Yaskawa INFORM job: CALIBRATION_RELATIVE.JBI

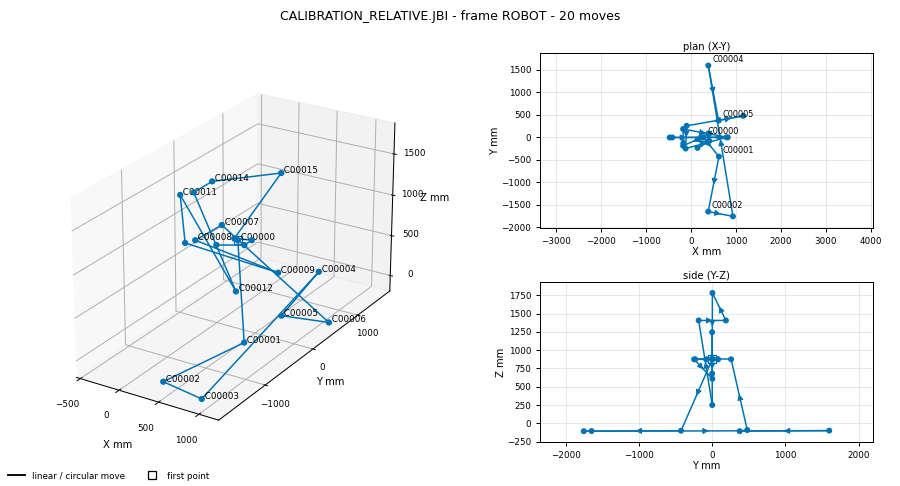
[picture p0: tool path of CALIBRATION_RELATIVE.JBI in frame ROBOT, 20 of 20 moves have a stored position in this frame; points joined in program order, loops and branches not executed]
/JOB
//NAME CALIBRATION_RELATIVE
//POS
///NPOS 20,0,0,0,0,0
///TOOL 0
///POSTYPE ROBOT
///RECTAN
///RCONF 1,0,0,0,0,0,0,0,0,0,0,0,0,0,0,0,0,0,0,0,0,0,0,0
C00000=274.980,-0.008,875.000,179.9989,44.9997,0.0020
C00001=622.573,-426.393,-101.139,-179.2940,-0.1745,-16.1282
C00002=383.550,-1649.719,-105.735,-178.5001,0.5026,-41.4095
C00003=933.399,-1756.204,-107.506,-178.6315,0.5025,-41.3677
C00004=385.503,1598.413,-99.610,-179.5797,-0.3013,-6.9319
C00005=613.623,374.870,-107.125,-179.5061,-0.2696,-6.9262
C00006=1163.774,478.153,-91.819,-179.4694,-0.2982,-6.9135
C00007=-96.141,257.633,874.999,180.0000,45.0002,110.4650
C00008=-118.644,-248.076,874.999,180.0000,45.0002,-115.5590
C00009=790.609,1.376,608.986,179.1795,83.3199,-0.7822
///RCONF 1,0,1,0,0,0,0,0,0,0,0,0,0,0,0,0,0,0,0,0,0,0,0,0
C00010=-414.668,-1.854,679.993,-179.8858,-2.8354,0.0446
C00011=-472.496,-2.009,1245.133,-179.8243,-31.5756,0.0258
///RCONF 1,0,0,0,0,0,0,0,0,0,0,0,0,0,0,0,0,0,0,0,0,0,0,0
C00012=249.873,-0.073,250.348,0.7052,79.6569,-179.2402
C00013=-173.865,-186.177,1406.145,147.2368,-45.5002,-134.7207
C00014=-174.385,186.529,1405.578,-146.8336,-45.3818,134.7676
///RCONF 0,0,0,0,0,0,0,0,0,0,0,0,0,0,0,0,0,0,0,0,0,0,0,0
C00015=818.445,1.458,1781.947,-6.0107,-88.9505,-173.7227
///RCONF 1,0,0,0,0,0,0,0,0,0,0,0,0,0,0,0,0,0,0,0,0,0,0,0
C00016=229.198,-0.125,884.124,179.9802,49.6969,-0.0171
///RCONF 1,0,0,0,1,0,0,0,0,0,0,0,0,0,0,0,0,0,0,0,0,0,0,0
C00017=404.652,79.634,874.999,179.9998,44.9999,-118.1512
C00018=406.759,-76.550,874.999,-179.9998,44.9999,118.4297
///RCONF 1,0,0,0,0,0,0,0,0,0,0,0,0,0,0,0,0,0,0,0,0,0,0,0
C00019=145.602,-233.286,874.998,180.0000,45.0007,-58.0294
//INST
///DATE 2026/08/24 08:52
///ATTR SC,RW,RJ
////FRAME ROBOT
///GROUP1 RB1
NOP
'1 HOME POSTION
MOVL C00000 V=423.3
'2 UF#2 S1 ORG
MOVL C00001 V=423.3
'3 UF#2 S1 RXX
MOVL C00002 V=423.3
'4 UF#2 S1 RXY
MOVL C00003 V=423.3
'5 UF#3 S2 ORG
MOVL C00004 V=423.3
'6 UF#3 S2 RXX
MOVL C00005 V=423.3
'7 UF#3 S2 RXY
MOVL C00006 V=423.3
'8 S+ SAFE LIMIT FROM HOME
MOVL C00007 V=423.3
'9 S- SAFE LIMIT FROM HOME
MOVL C00008 V=423.3
'10 L+ SAFE LIMIT FROM HOME
MOVL C00009 V=423.3
'11 L- SAFE LIMIT FROM HOME
MOVL C00010 V=423.3
'12 U+ SAFE LIMIT FROM HOME
MOVL C00011 V=423.3
'13 U- SAFE LIMIT FROM HOME
MOVL C00012 V=423.3
'14 R+ SAFE LIMIT FROM HOME
MOVL C00013 V=423.3
'15 R- SAFE LIMIT FROM HOME
MOVL C00014 V=423.3
'16 B+ SAFE LIMIT FROM HOME
MOVL C00015 V=423.3
'17 B- SAFE LIMIT FROM HOME
MOVL C00016 V=423.3
'18 T+ SAFE LIMIT FROM HOME
MOVL C00017 V=423.3
'19 T- SAFE LIMIT FROM HOME
MOVL C00018 V=423.3
'20 EXTRA CLEAR POSE
MOVL C00019 V=423.3
END
